// Mitsubishi GX Works2 project: PLC_Group10   PLC: FX3G

// global labels: Global1
VAR_GLOBAL
  ST_DAY10 AT X010 : BOOL;  (* מתג פולס בעליה שמטרתו להתחיל את היום *)
  O_Stock AT D1108 : REAL;  (* תפוזים במלאי *)
  P_Stock AT D1112 : REAL;  (* פומלות במלאי *)
  WashFruit AT X002 : BOOL;  (* מתג תחילת שטיפת הפירות *)
END_VAR
VAR_GLOBAL CONSTANT
  TVal : INT := 30;  (* ערך 3 שניות *)
END_VAR
VAR_GLOBAL
  Coil_Timer1 AT TC3 : BOOL;  (* טיימר 3 שניות להדלקת נורה Y5 *)
  End_CoilT1 AT TS3 : BOOL;  (* מתג שנפתח לאחר 3 שניות *)
  Start_Wash AT Y005 : BOOL;  (* נורה עבור תחילת שלב השטיפה *)
  C_WashM AT D1116 : REAL;  (* קלמנטינות בכלי שטיפה *)
END_VAR
VAR_GLOBAL CONSTANT
  Const05 : REAL := 0.5;  (* קבוע 0.5 להכפלת כמות התפוזים על פי תנאי לתחילת עבודה *)
END_VAR
VAR_GLOBAL
  End_Day AT M7 : BOOL;  (* משתנה נורת עזר 7-סיום עבודה *)
  All_Day_On AT Y010 : BOOL;  (* נורה שדולקת לאורך כל היום *)
END_VAR
VAR_GLOBAL CONSTANT
  Zero : REAL;  (* קבוע אפס *)
END_VAR
VAR_GLOBAL
  Val_Bool AT M1 : BOOL;  (* נורת חיווי שבודקת אם הקלט הוא אפס *)
  Validation_Check AT M0 : BOOL;  (* נורת חיווי תחילת הרצה *)
  O_WashM AT D1118 : REAL;  (* תפוזים בכלי שטיפה *)
  P_WashM AT D1120 : REAL;  (* פומלות בכלי שטיפה *)
END_VAR
VAR_GLOBAL CONSTANT
  Const2 : INT := 2;  (* בדיקת כמות תפוזים *)
END_VAR
VAR_GLOBAL
  Can_Start_Valid AT M8 : BOOL;  (* בדיקת כמות תפוזים במלאי *)
  Start_3sec AT M9 : BOOL;  (* נורת חיווי תחילת טיימר 3 שניות *)
  Half_Oranges AT D1126 : REAL;  (* חצי מכמות התפוזים במלאי *)
END_VAR
VAR_GLOBAL CONSTANT
  Max_Orange100 : INT := 100;  (* כמות מקסימלית של תפוזים בשטיפה *)
END_VAR
VAR_GLOBAL
  Orange_AmountInWash AT D1128 : REAL;  (* כמות התפוזים לשטיפה *)
  Start_Check AT X003 : BOOL;  (* מתג תחילת בדיקת איכות מיץ *)
  Start_Sq AT X001 : BOOL;  (* תחילת סחיטת הפירות *)
  Sq_Light AT Y001 : BOOL;  (* נורת סחיטת הפירות *)
  allToSq AT D1130 : REAL;  (* העברת פירות למיכל סחיטה *)
  Sq_Tank AT D1132 : REAL;  (* מיכל סחיטת הפירות *)
  Moved_To_Sq AT M12 : BOOL;  (* הפירות הועברו למיכל הסחיטה *)
END_VAR
VAR_GLOBAL CONSTANT
  C_Wash_Reset : REAL;  (* איפוס מיכל השטיפה של הקלמנטינות *)
  O_Wash_Reset : REAL;  (* איפוס מיכל השטיפה של התפוזים *)
  P_Wash_Reset : REAL;  (* איפוס מיכל השטיפה של הפומלות *)
END_VAR
VAR_GLOBAL
  Moved_To_Wash AT M13 : BOOL;  (* סיום העברת הפירות למיכלי השטיפה *)
  Sq_LightM AT M14 : BOOL;  (* חיווי נורת סחיטת הפירות *)
  P_C_Wash_Amount AT D1110 : REAL;  (* מספר קלמנטינות ופומלות שיעבור למיכל השטיפה *)
  O_InWash AT M17 : BOOL;  (* חיווי של מספר התפוזים לשטיפה *)
  Min_P_C AT M16 : BOOL;  (* כמות הקלנטינות והפומלות שיכנסו למיכל השטיפה *)
  Min_O AT M15 : BOOL;  (* כמות התפוזים שיכנסו למיכל השטיפה *)
  Stop_SqLight AT M11 : BOOL;  (* כיבוי נורת סחיטת הפירות *)
  Start_3sec_Sq AT X011 : BOOL;  (* מתג הדלקת הבהוב 3 שניות *)
  Click_Twice AT CC1 : BOOL;  (* מונה אירועים שמחכה לשתי לחיצות על מתג איקס 11 *)
END_VAR
VAR_GLOBAL CONSTANT
  Counter_2Clicks : INT := 2;  (* 2לחיצות על איקס 11 *)
END_VAR
VAR_GLOBAL
  Timer_All_Sq AT TC36 : BOOL;  (* טיימר סחיטת פירות למשך 3שניות *)
END_VAR
VAR_GLOBAL CONSTANT
  Val_3Sec : INT := 30;  (* טיימר עובד למשך 3 שניות *)
END_VAR
VAR_GLOBAL
  End_Counting AT CS1 : BOOL;  (* לאחר 2 לחיצות מתחילה הסחיטה *)
  Reset_Flickering AT M31 : BOOL;  (* משתנה שמאתחל את פונקציית ההבהוב *)
  Timer_Sq_Y2 AT TC30 : BOOL;  (* טיימר סחיטת פירות למשך 3שניות *)
END_VAR
VAR_GLOBAL CONSTANT
  Half_sec : INT := 5;  (* נורה וואי 2 דולקת למשך חצי דקה *)
END_VAR
VAR_GLOBAL
  Start_Y2 AT TS30 : BOOL;  (* הדלקת נורה Y2 *)
  Light_Y2 AT Y002 : BOOL;  (* נורת הבהוב Y2 *)
  Timer_Sq_Y3 AT TC32 : BOOL;  (* טיימר שמפעיל את וואי3 שתהבהב *)
  Start_Y3 AT TS32 : BOOL;  (* הדלקת נורה Y3 *)
  Light_Y3 AT Y003 : BOOL;  (* נורת הבהוב Y3 *)
  Stop_Timer_3Sec AT TS36 : BOOL;  (* מפסיק הבהוב לאחר 3 שניות *)
  Juice_Cont AT D4000 : REAL;  (* מיכל מיץ *)
  Moved_To_Juice AT M37 : BOOL;  (* הועברו הפירות הסחוטים למיכל המיץ *)
  Start_Read_Analog AT M40 : BOOL;  (* נורת עזר- יכול לבדוק את הקלט האנלוגי *)
  Analog_Input2 AT D8281 : INT;  (* האינפוט האנלוגי *)
  Analog_Value AT D8291 : REAL;  (* הערך האנאלוגי *)
END_VAR
VAR_GLOBAL CONSTANT
  Const01 : REAL := 1.0;  (* קבוע 1- חסם תחתון לבדיקת איכות תקינה *)
END_VAR
VAR_GLOBAL
  Counting_Input AT CC2 : BOOL;  (* סופר מספר ניסיונות לקלט *)
END_VAR
VAR_GLOBAL CONSTANT
  Two_Inputs : INT := 2;  (* 2 אופצית להכנסת קלט *)
END_VAR
VAR_GLOBAL
  Two_Invalid_Counted AT CS2 : BOOL;  (* נספרו 2 קלטים מחוץ לטווח *)
  Start_5sec AT M42 : BOOL;  (* נורת חיווי תחילת טיימר 5 שניות *)
  Coil_Timer_5sec AT TC34 : BOOL;  (* Y4 תדלוק למשך 5 שניות *)
END_VAR
VAR_GLOBAL CONSTANT
  T_Value_5sec : INT := 50;  (* ערך 5 שניות *)
END_VAR
VAR_GLOBAL
  Finished_5sec AT M43 : BOOL;  (* נורת עזר- סיום 5 שניות *)
  End_CoilT2 AT TS34 : BOOL;  (* מתג שנפתח לאחר 5 שניות *)
  Finish_Qcheck AT Y004 : BOOL;  (* נורה שבדיקת האיכות בוצעה בהצלחה *)
  Storage_Cont AT D4002 : REAL;  (* מיכל אחסון *)
  Moved_To_Storage AT M44 : BOOL;  (* הועבר המיץ למיכל האחסון *)
  Empty_Sq_Tank AT M45 : BOOL;  (* המיץ הועבר ממיכל הסחיטה למיכל המיץ *)
END_VAR
VAR_GLOBAL CONSTANT
  Convert_Analog : REAL := 404.5;  (* המרת ערך אנאלוגי מהבקר למחשב *)
  Const5 : REAL := 5.0;  (* קבוע 5 *)
END_VAR
VAR_GLOBAL
  Input_Not_In_Range_1 AT M5 : BOOL;  (* נורת עזר- הקלט האנלוגי לא בטווח- קטן מ1 *)
  Input_Not_In_Range_5 AT M6 : BOOL;  (* נורת עזר- הקלט האנלוגי לא בטווח- גדול מ5 *)
  M_Start_Check AT M3 : BOOL;  (* נורת חיווי שמתג X3 הופעל *)
  Input_In_Range AT M4 : BOOL;  (* נורת עזר- הקלט האנלוגי בטווח *)
  End_Day_007 AT X007 : BOOL;  (* מתג סיום יום העבודה *)
  Not_In_Range_5 AT M49 : BOOL;  (* הערך גדול מ5 *)
  Not_In_Range_1 AT M47 : BOOL;  (* הערך קטן מ1 *)
  End_Day_Flickering AT TC38 : BOOL;  (* תחילת הבהוב סיום יום העבודה *)
  Flickering_End_Day AT TC40 : BOOL;  (* הבהוב סוף יום *)
  End_3Sec_End_Day AT TS38 : BOOL;  (* סיום הבהוב 3 שניות סוף יום *)
  End_Half_Sec AT TS40 : BOOL;  (* סיום חצי שניה של הבהוב *)
  Start_Half_Sec AT M50 : BOOL;  (* תחילת חצי שניה *)
  Continue_To_Blink AT M51 : BOOL;  (* המשך הבהוב *)
  Help_Timer_Half_Sec AT TC41 : BOOL;  (* טיימר חצי שניה *)
  Help_End_Half_Sec AT TS41 : BOOL;  (* סיום חצי שניה של הבהוב עזרה *)
  Help_Me AT M52 : BOOL;  (* הצילינינא *)
  Help_Me_2 AT M53 : BOOL;  (* הצילינינא2 *)
  No_More AT M55 : BOOL;  (* סיום עבודה *)
END_VAR
VAR_GLOBAL CONSTANT
  Const_4 : REAL := 4.0;  (* קבוע 4- כמות מיץ מינימלית להמשך תהליך *)
END_VAR
VAR_GLOBAL
  Move_To_Filter AT M56 : BOOL;  (* נורת עזר- 4 ליטר מיץ הועבר למיכל הסינון *)
  Juice_To_Filter AT D1102 : REAL;  (* העברת 4 ליטר מיץ למיכל סינון *)
  Start_Filtering AT X000 : BOOL;  (* מתג שמתחיל את שלב הסינון *)
  Juice_Filtered AT D1124 : REAL;  (* מיכל מיץ מסונן *)
  Storage_Filtered AT M57 : BOOL;  (* נורת עזר- הורדת המיץ המסונן מהאחסון *)
  Aperol_Spritz AT D4004 : REAL;  (* אפרול שפריץ- המיץ המסונן האלכוהולי שלנו *)
  Analog_Output AT D8282 : INT;  (* האאוטפוט האנלוגי *)
  Filtering_Time AT Y000 : BOOL;  (* נורה שדולקת בכל תהליך הסינון *)
END_VAR
VAR_GLOBAL CONSTANT
  Two_Liter_Alcohol : REAL := 2.0;  (* הוספת 2 ליטר אלכוהול למיץ המסונן *)
END_VAR
VAR_GLOBAL
  Aperol_To_Taste AT Y006 : BOOL;  (* נורה שנדלקת כשהאפרול מוכן *)
  Counting_Rates AT CC3 : BOOL;  (* סופר 4 ציונים *)
END_VAR
VAR_GLOBAL CONSTANT
  Four_Rates : INT := 4;  (* 4 ציונים *)
END_VAR
VAR_GLOBAL
  Four_Rates_Given AT CS3 : BOOL;  (* ניתנו 4 ציונים *)
  Start_Rating AT X005 : BOOL;  (* מתג שמתחיל קליטת ציון *)
  M_Start_Check_Rate AT M10 : BOOL;  (* נורת חיווי ניתן ציון *)
  Read_Analog_Rate AT M18 : BOOL;  (* נורת עזר- יכול לבדוק את הקלט האנלוגי *)
  Analog_Value_Rate AT D8293 : REAL;  (* הערך האנאלוגי *)
  Total_Rates AT D1114 : REAL;  (* סך הציונים *)
  Average_Grade AT D1106 : INT;  (* הציון הממוצע של המשקה *)
  Final_Grade AT M59 : BOOL;  (* חושב ציון סופי למשקה *)
  Analog_Input1 AT D8280 : INT;  (* האינפוט האנלוגי *)
  Analog_Showed AT M30 : BOOL;  (* הציון נמצאבOUTPUT *)
  Total_Rates_W AT D1122 : INT;  (* סך הציונים בWORLD *)
  End_Filtering_Light AT TS50 : BOOL;  (* סיום נורת הסינון *)
  Start_Filtering_Light AT TC50 : BOOL;  (* מתג שמתחיל את שלב הסינון *)
  Drink_Is_Ready AT M28 : BOOL;  (* המשקה האלכוהולי מוכן! *)
  Drink_Timer AT TC60 : BOOL;  (* טיימר משקה הוכן *)
END_VAR
VAR_GLOBAL CONSTANT
  Four_Sec : INT := 40;  (* 4 שניות *)
END_VAR
VAR_GLOBAL
  Moved_From_Storage AT M26 : BOOL;  (* העברה 4 מהאחסון לסינון *)
  Average_Output AT D1134 : INT;  (* ממוצע להצגה לאאוטפוט *)
  Output_Convert AT M32 : BOOL;  (* המרה לאאוטפוט *)
  Grade_Added AT M39 : BOOL;  (* נוסף ציון *)
  Lets_Get_Wasted AT M46 : BOOL;  (* יאללה פארטי *)
END_VAR
VAR_GLOBAL CONSTANT
  Const400 : INT := 400;  (* הכפלת אפרול שפריץ בקבוע בשביל שיוציא באנלוג אאוטפוט *)
END_VAR
VAR_GLOBAL
  If_Fruits_Ended AT M24 : BOOL;  (* נגמר סוג אחד או יותר של פרי *)
  Drink_Timer_Ended AT TS60 : BOOL;  (* סיום טיימר נורת ערבוב *)
  Start_Again AT M60 : BOOL;  (* סיום יום והתחלת יום חדש *)
  Did_You_Get_True AT M88 : BOOL;  (* נורה שבודקת שעבר זרם דרך בדיקת שני תפוזים *)
  End_Day_Bulb AT M70 : BOOL;  (* מתג סיום יום העבודה *)
  C_Stock AT D4006 : REAL;  (* קלמנטינות במלאי *)
  Damaged_Juice AT M73 : BOOL;  (* מיץ לא תקין *)
END_VAR

// task Task_01 (event TRUE, interval 0, priority 31): POU_01

PROGRAM POU_01
VAR
  O_output : REAL;
  C_output : REAL;
  P_output : REAL;
  Start_Flickering : BOOL;  (* תחילת שלב הסחיטה- ההבהוב *)
  Move_To : BOOL;
END_VAR
(* structured ladder/FBD written out as ST: instructions are called as NAME(EN, inputs, outputs); _pN, _eN, _tN stand for wires *)
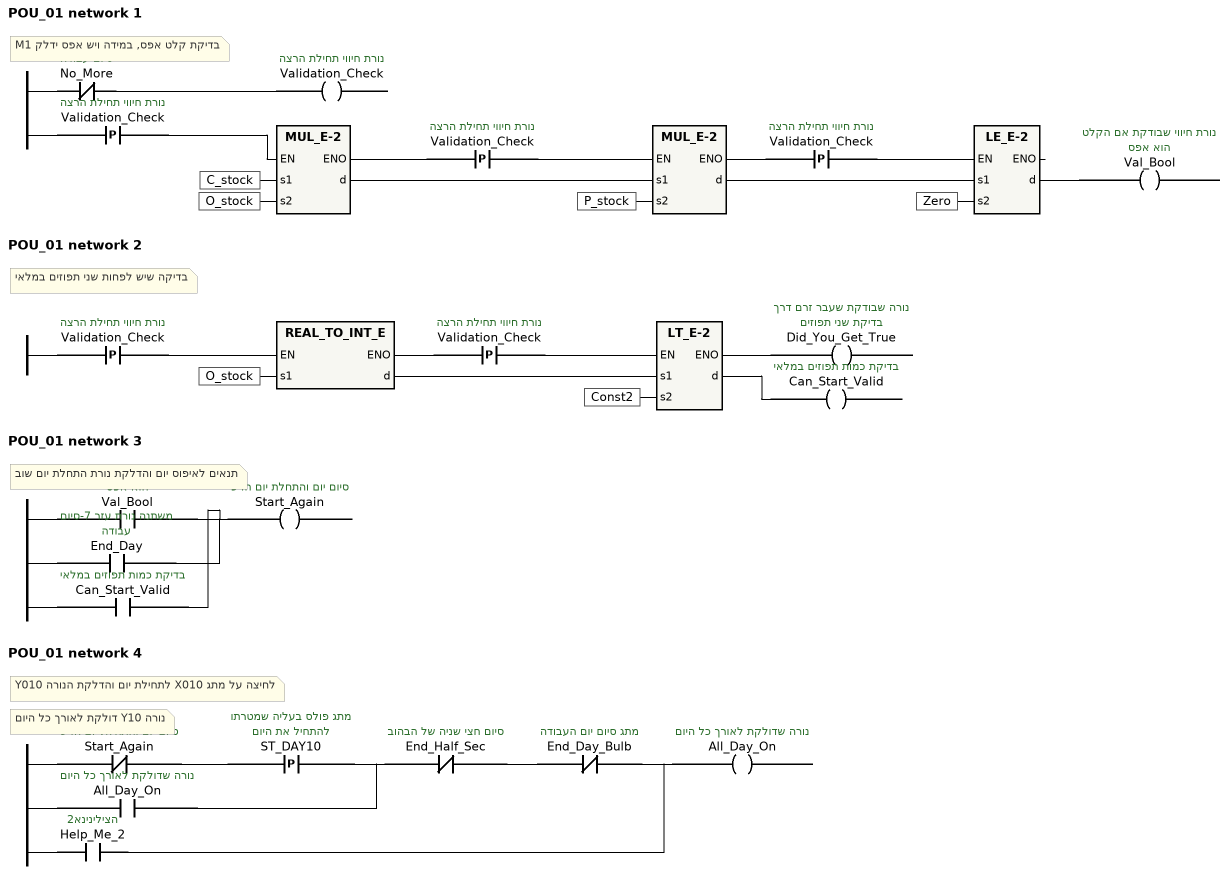
(* network 1 *)
(* בדיקת קלט אפס, במידה ויש אפס ידלק M1 *)
Validation_Check := NOT No_More;
_e2 := MUL_E(LDP(TRUE, Validation_Check), C_stock, O_stock, _t1);
_e4 := MUL_E(_e2 AND LDP(TRUE, Validation_Check), _t1, P_stock, _t3);
LE_E(_e4 AND LDP(TRUE, Validation_Check), _t3, Zero, _t5);
Val_Bool := _t5;
(* network 2 *)
(* בדיקה שיש לפחות שני תפוזים במלאי *)
_e2 := REAL_TO_INT_E(LDP(TRUE, Validation_Check), O_stock, _t1);
_e4 := LT_E(_e2 AND LDP(TRUE, Validation_Check), _t1, Const2, _t3);
Did_You_Get_True := _e4;
Can_Start_Valid := _t3;
(* network 3 *)
(* תנאים לאיפוס יום והדלקת נורת התחלת יום שוב *)
Start_Again := Val_Bool OR End_Day OR Can_Start_Valid;
(* network 4 *)
(* לחיצה על מתג X010 לתחילת יום והדלקת הנורה Y010 *)
(* נורה Y10 דולקת לאורך כל היום *)
All_Day_On := ((((NOT Start_Again AND LDP(TRUE, ST_DAY10)) OR All_Day_On) AND NOT End_Half_Sec) AND NOT End_Day_Bulb) OR Help_Me_2;
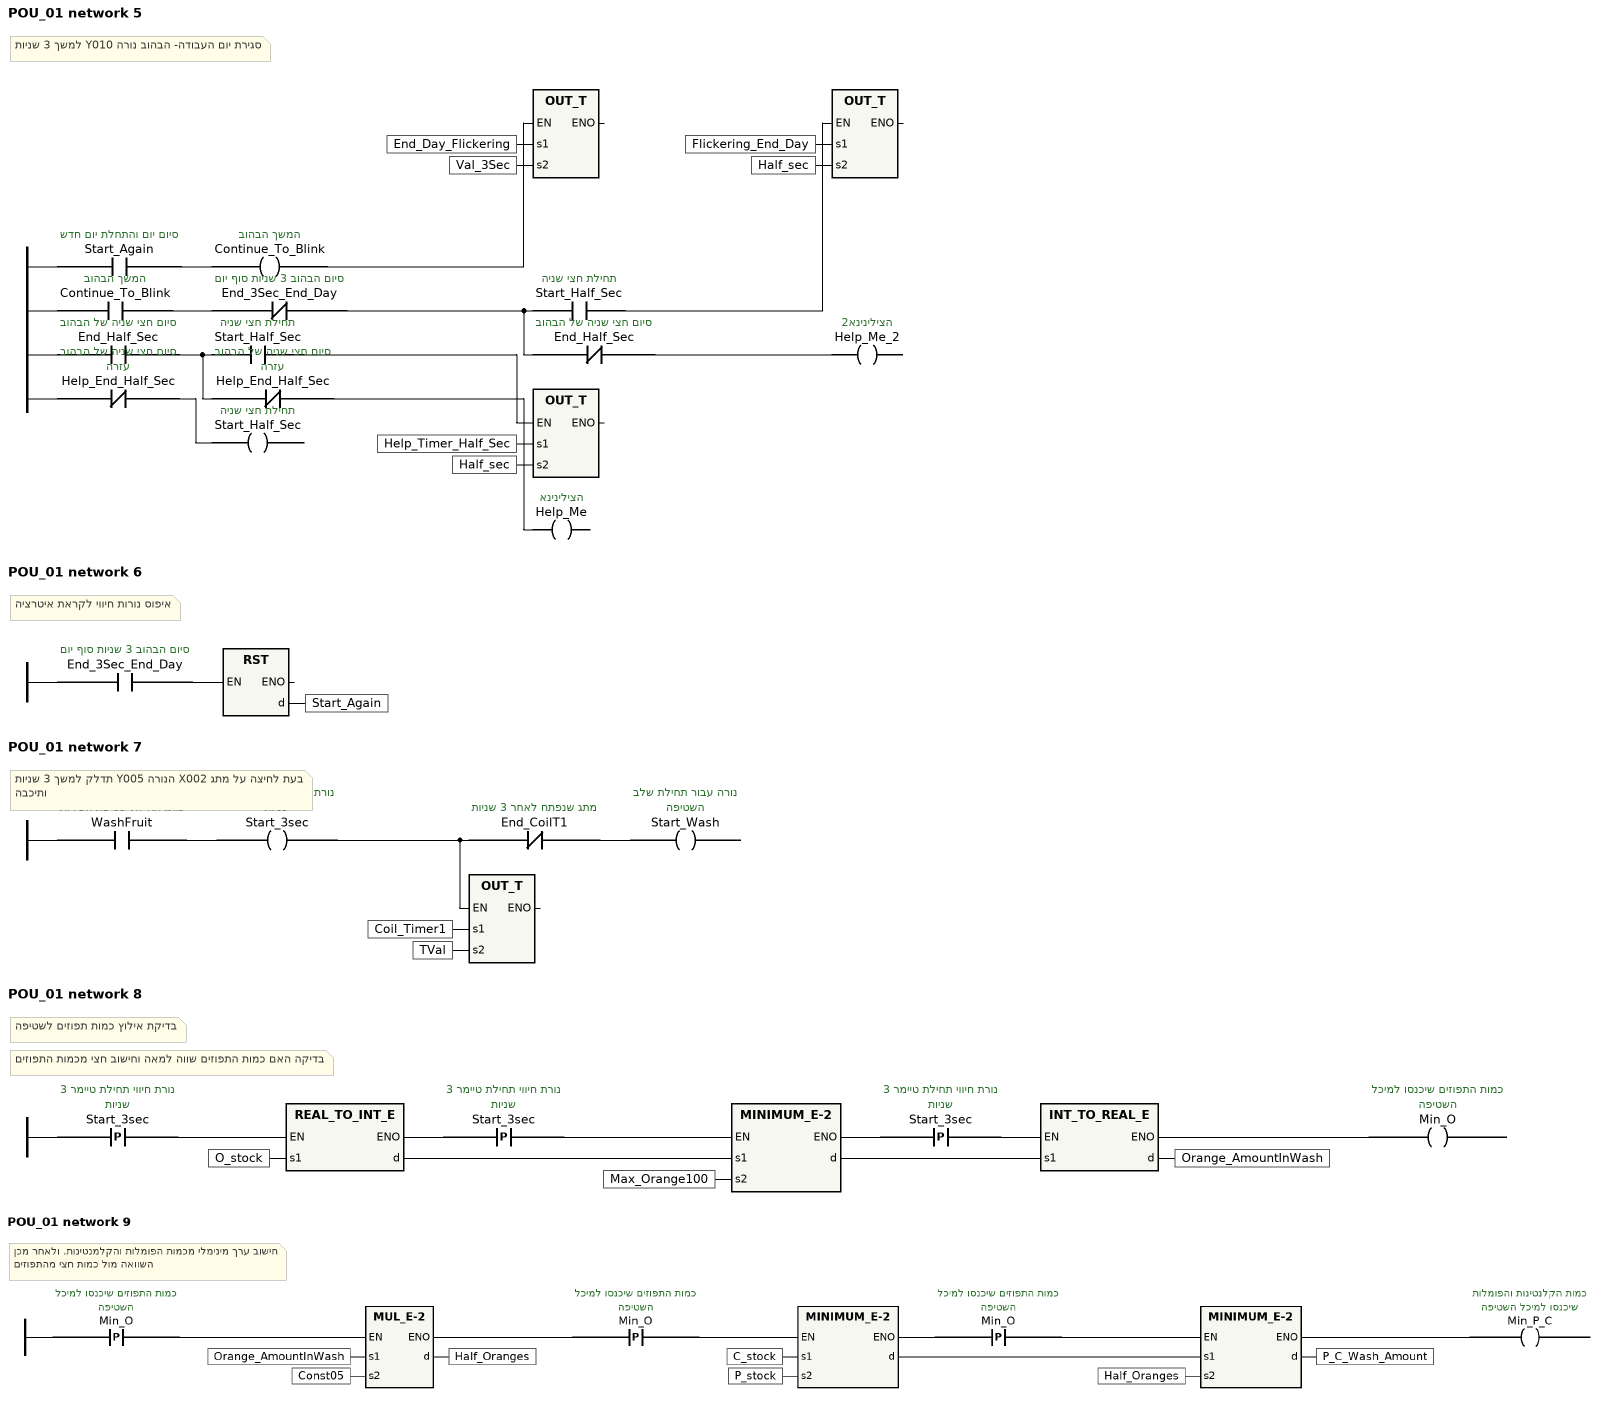
(* network 5 *)
(* סגירת יום העבודה- הבהוב נורה Y010 למשך 3 שניות *)
Continue_To_Blink := Start_Again;
OUT_T(Start_Again, End_Day_Flickering, Val_3Sec);
_p1 := Continue_To_Blink AND NOT End_3Sec_End_Day;
OUT_T(_p1 AND Start_Half_Sec, Flickering_End_Day, Half_sec);
Help_Me_2 := _p1 AND NOT End_Half_Sec;
OUT_T(End_Half_Sec AND Start_Half_Sec, Help_Timer_Half_Sec, Half_sec);
Help_Me := End_Half_Sec AND NOT Help_End_Half_Sec;
Start_Half_Sec := NOT Help_End_Half_Sec;
(* network 6 *)
(* איפוס נורות חיווי לקראת איטרציה *)
RST(End_3Sec_End_Day, Start_Again);
(* network 7 *)
(* בעת לחיצה על מתג X002 הנורה Y005 תדלק למשך 3 שניות ותיכבה *)
Start_3sec := WashFruit;
Start_Wash := WashFruit AND NOT End_CoilT1;
OUT_T(WashFruit, Coil_Timer1, TVal);
(* network 8 *)
(* בדיקת אילוץ כמות תפוזים לשטיפה *)
(* בדיקה האם כמות התפוזים שווה למאה וחישוב חצי מכמות התפוזים *)
_e2 := REAL_TO_INT_E(LDP(TRUE, Start_3sec), O_stock, _t1);
_e4 := MINIMUM_E(_e2 AND LDP(TRUE, Start_3sec), _t1, Max_Orange100, _t3);
_e5 := INT_TO_REAL_E(_e4 AND LDP(TRUE, Start_3sec), _t3, Orange_AmountInWash);
Min_O := _e5;
(* network 9 *)
(* חישוב ערך מינימלי מכמות הפומלות והקלמנטינות. ולאחר מכן השוואה מול כמות חצי מהתפוזים *)
_e1 := MUL_E(LDP(TRUE, Min_O), Orange_AmountInWash, Const05, Half_Oranges);
_e3 := MINIMUM_E(_e1 AND LDP(TRUE, Min_O), C_stock, P_stock, _t2);
_e4 := MINIMUM_E(_e3 AND LDP(TRUE, Min_O), _t2, Half_Oranges, P_C_Wash_Amount);
Min_P_C := _e4;
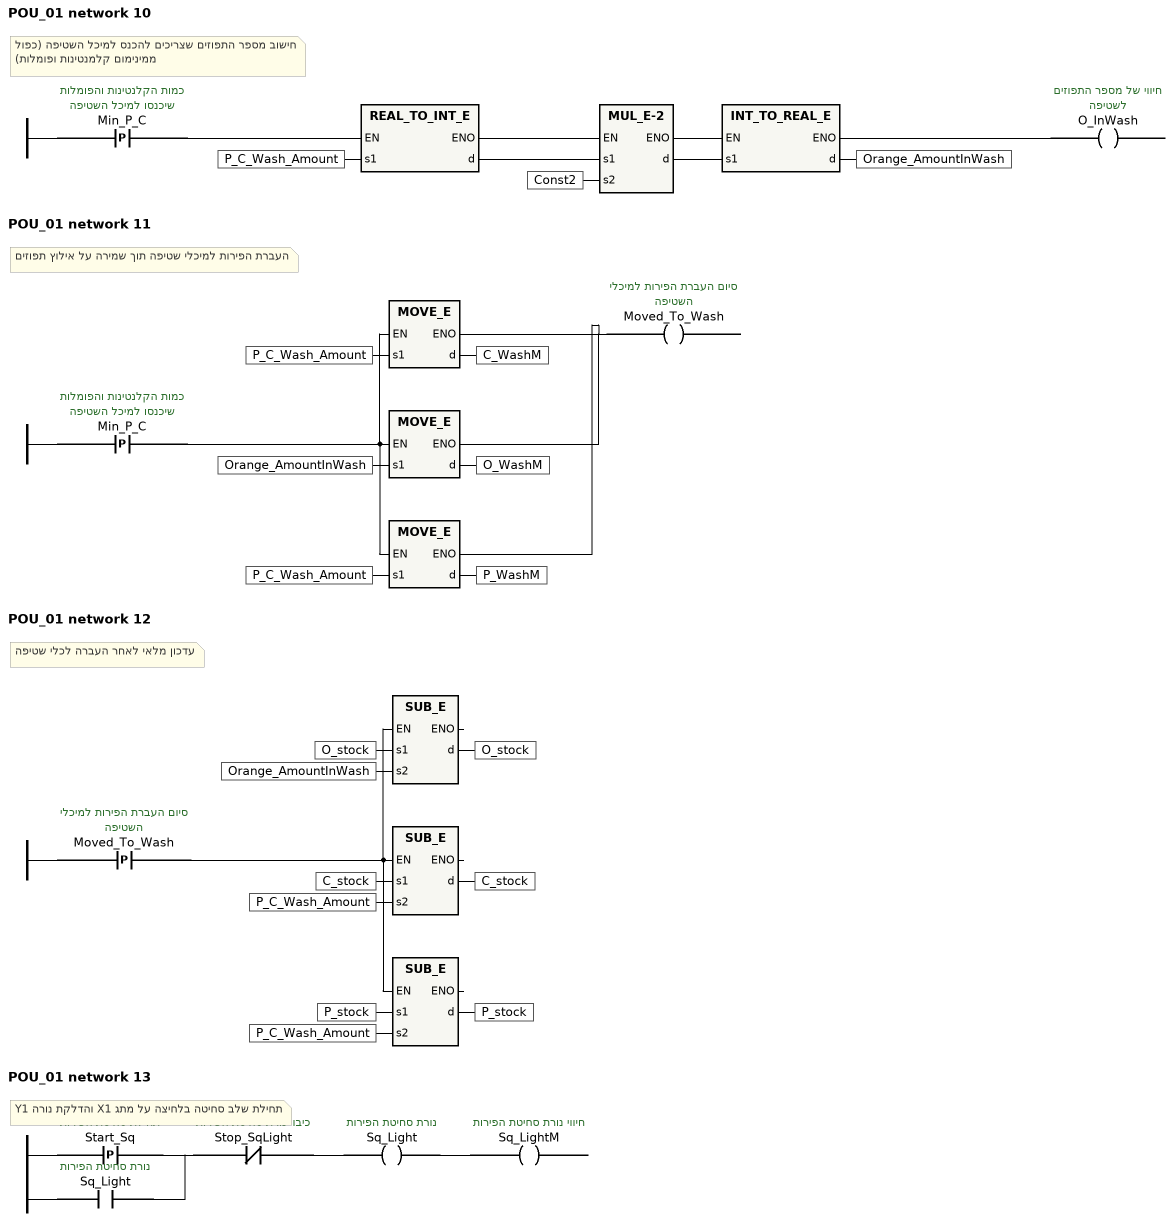
(* network 10 *)
(* חישוב מספר התפוזים שצריכים להכנס למיכל השטיפה (כפול ממינימום קלמנטינות ופומלות) *)
_e2 := REAL_TO_INT_E(LDP(TRUE, Min_P_C), P_C_Wash_Amount, _t1);
_e4 := MUL_E(_e2, _t1, Const2, _t3);
_e5 := INT_TO_REAL_E(_e4, _t3, Orange_AmountInWash);
O_InWash := _e5;
(* network 11 *)
(* העברת הפירות למיכלי שטיפה תוך שמירה על אילוץ תפוזים *)
_p1 := LDP(TRUE, Min_P_C);
_e2 := MOVE_E(_p1, P_C_Wash_Amount, C_WashM);
_e3 := MOVE_E(_p1, Orange_AmountInWash, O_WashM);
_e4 := MOVE_E(_p1, P_C_Wash_Amount, P_WashM);
Moved_To_Wash := _e2 OR _e3 OR _e4;
(* network 12 *)
(* עדכון מלאי לאחר העברה לכלי שטיפה *)
_p1 := LDP(TRUE, Moved_To_Wash);
SUB_E(_p1, O_stock, Orange_AmountInWash, O_stock);
SUB_E(_p1, C_stock, P_C_Wash_Amount, C_stock);
SUB_E(_p1, P_stock, P_C_Wash_Amount, P_stock);
(* network 13 *)
(* תחילת שלב סחיטה בלחיצה על מתג X1 והדלקת נורה Y1 *)
_p1 := (LDP(TRUE, Start_Sq) OR Sq_Light) AND NOT Stop_SqLight;
Sq_Light := _p1;
Sq_LightM := _p1;
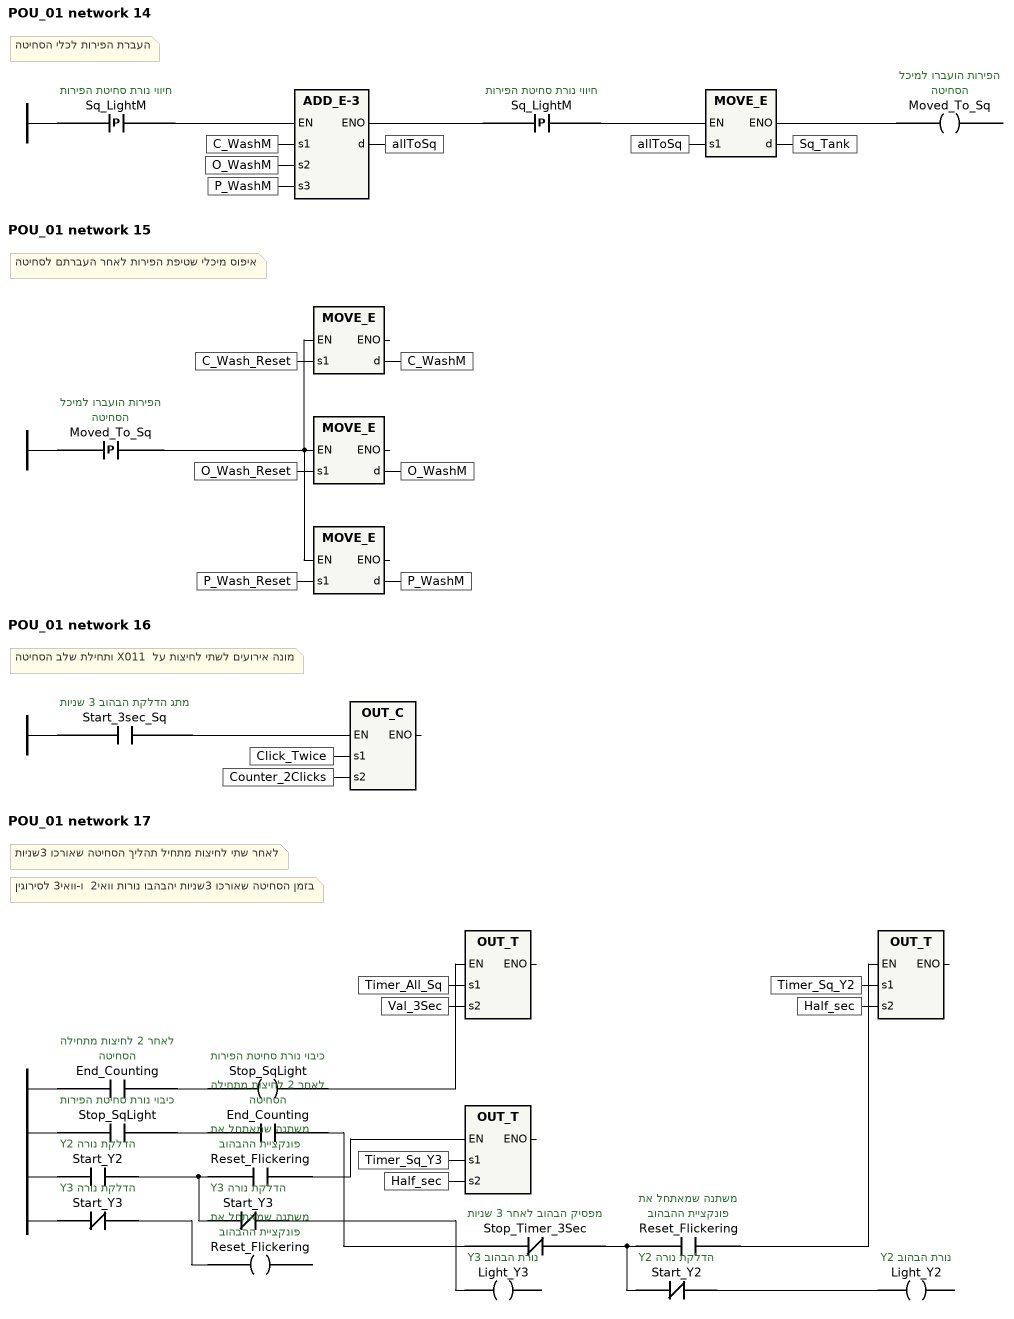
(* network 14 *)
(* העברת הפירות לכלי הסחיטה *)
_e1 := ADD_E(LDP(TRUE, Sq_LightM), C_WashM, O_WashM, P_WashM, allToSq);
_e2 := MOVE_E(_e1 AND LDP(TRUE, Sq_LightM), allToSq, Sq_Tank);
Moved_To_Sq := _e2;
(* network 15 *)
(* איפוס מיכלי שטיפת הפירות לאחר העברתם לסחיטה *)
_p1 := LDP(TRUE, Moved_To_Sq);
MOVE_E(_p1, C_Wash_Reset, C_WashM);
MOVE_E(_p1, O_Wash_Reset, O_WashM);
MOVE_E(_p1, P_Wash_Reset, P_WashM);
(* network 16 *)
(* מונה אירועים לשתי לחיצות על  X011 ותחילת שלב הסחיטה *)
OUT_C(Start_3sec_Sq, Click_Twice, Counter_2Clicks);
(* network 17 *)
(* לאחר שתי לחיצות מתחיל תהליך הסחיטה שאורכו 3שניות *)
(* בזמן הסחיטה שאורכו 3שניות יהבהבו נורות וואי2  ו-וואי3 לסירוגין *)
Stop_SqLight := End_Counting;
OUT_T(End_Counting, Timer_All_Sq, Val_3Sec);
_p1 := Stop_SqLight AND End_Counting AND NOT Stop_Timer_3Sec;
OUT_T(_p1 AND Reset_Flickering, Timer_Sq_Y2, Half_sec);
Light_Y2 := _p1 AND NOT Start_Y2;
OUT_T(Start_Y2 AND Reset_Flickering, Timer_Sq_Y3, Half_sec);
Light_Y3 := Start_Y2 AND NOT Start_Y3;
Reset_Flickering := NOT Start_Y3;
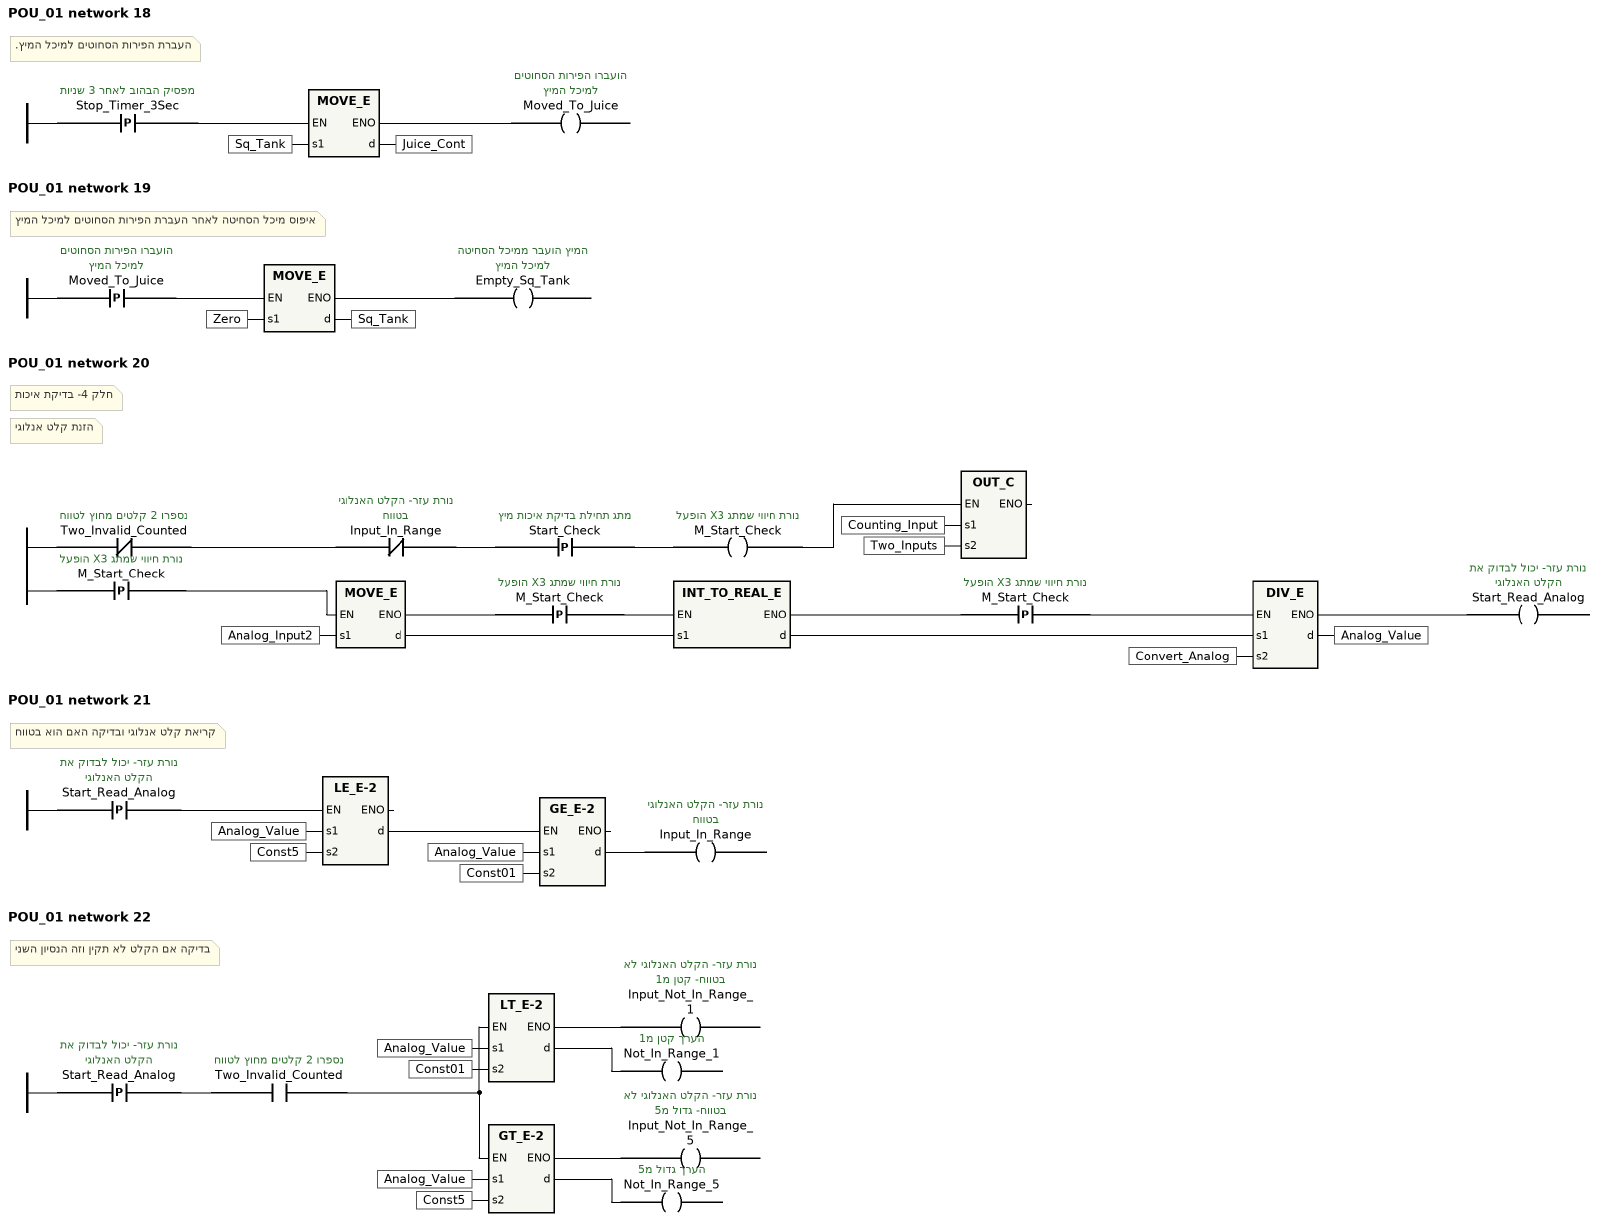
(* network 18 *)
(* העברת הפירות הסחוטים למיכל המיץ. *)
_e1 := MOVE_E(LDP(TRUE, Stop_Timer_3Sec), Sq_Tank, Juice_Cont);
Moved_To_Juice := _e1;
(* network 19 *)
(* איפוס מיכל הסחיטה לאחר העברת הפירות הסחוטים למיכל המיץ *)
_e1 := MOVE_E(LDP(TRUE, Moved_To_Juice), Zero, Sq_Tank);
Empty_Sq_Tank := _e1;
(* network 20 *)
(* חלק 4- בדיקת איכות *)
(* הזנת קלט אנלוגי *)
_p1 := NOT Two_Invalid_Counted AND NOT Input_In_Range AND LDP(TRUE, Start_Check);
M_Start_Check := _p1;
OUT_C(_p1, Counting_Input, Two_Inputs);
_e3 := MOVE_E(LDP(TRUE, M_Start_Check), Analog_Input2, _t2);
_e5 := INT_TO_REAL_E(_e3 AND LDP(TRUE, M_Start_Check), _t2, _t4);
_e6 := DIV_E(_e5 AND LDP(TRUE, M_Start_Check), _t4, Convert_Analog, Analog_Value);
Start_Read_Analog := _e6;
(* network 21 *)
(* קריאת קלט אנלוגי ובדיקה האם הוא בטווח *)
LE_E(LDP(TRUE, Start_Read_Analog), Analog_Value, Const5, _t1);
GE_E(_t1, Analog_Value, Const01, _t2);
Input_In_Range := _t2;
(* network 22 *)
(* בדיקה אם הקלט לא תקין וזה הנסיון השני *)
_p1 := LDP(TRUE, Start_Read_Analog) AND Two_Invalid_Counted;
_e3 := LT_E(_p1, Analog_Value, Const01, _t2);
Input_Not_In_Range_1 := _e3;
Not_In_Range_1 := _t2;
_e5 := GT_E(_p1, Analog_Value, Const5, _t4);
Input_Not_In_Range_5 := _e5;
Not_In_Range_5 := _t4;
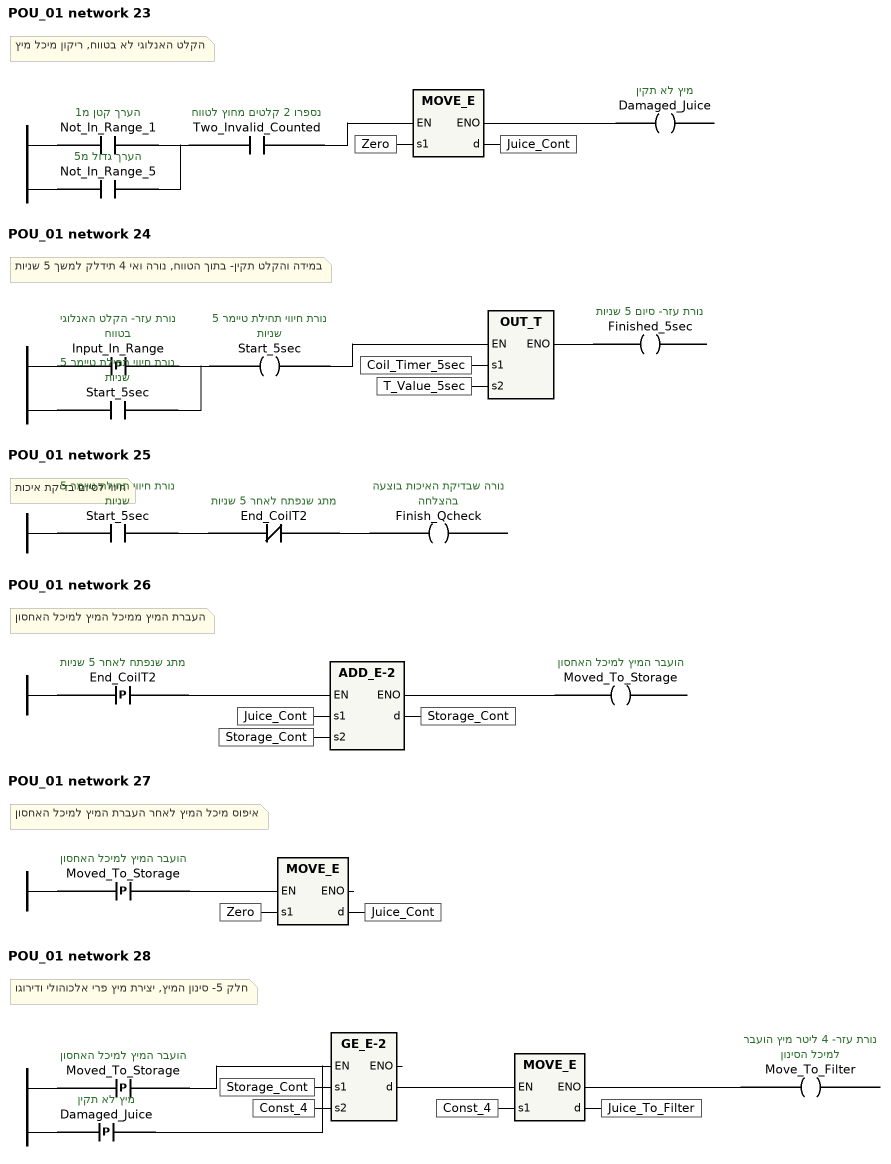
(* network 23 *)
(* הקלט האנלוגי לא בטווח, ריקון מיכל מיץ *)
_e1 := MOVE_E((Not_In_Range_1 OR Not_In_Range_5) AND Two_Invalid_Counted, Zero, Juice_Cont);
Damaged_Juice := _e1;
(* network 24 *)
(* במידה והקלט תקין- בתוך הטווח, נורה ואי 4 תידלק למשך 5 שניות *)
_p1 := LDP(TRUE, Input_In_Range) OR Start_5sec;
Start_5sec := _p1;
_e2 := OUT_T(_p1, Coil_Timer_5sec, T_Value_5sec);
Finished_5sec := _e2;
(* network 25 *)
(* חיווי לסיום בדיקת איכות *)
Finish_Qcheck := Start_5sec AND NOT End_CoilT2;
(* network 26 *)
(* העברת המיץ ממיכל המיץ למיכל האחסון *)
_e1 := ADD_E(LDP(TRUE, End_CoilT2), Juice_Cont, Storage_Cont, Storage_Cont);
Moved_To_Storage := _e1;
(* network 27 *)
(* איפוס מיכל המיץ לאחר העברת המיץ למיכל האחסון *)
MOVE_E(LDP(TRUE, Moved_To_Storage), Zero, Juice_Cont);
(* network 28 *)
(* חלק 5- סינון המיץ, יצירת מיץ פרי אלכוהולי ודירוגו *)
GE_E(LDP(TRUE, Moved_To_Storage) OR LDP(TRUE, Damaged_Juice), Storage_Cont, Const_4, _t1);
_e2 := MOVE_E(_t1, Const_4, Juice_To_Filter);
Move_To_Filter := _e2;
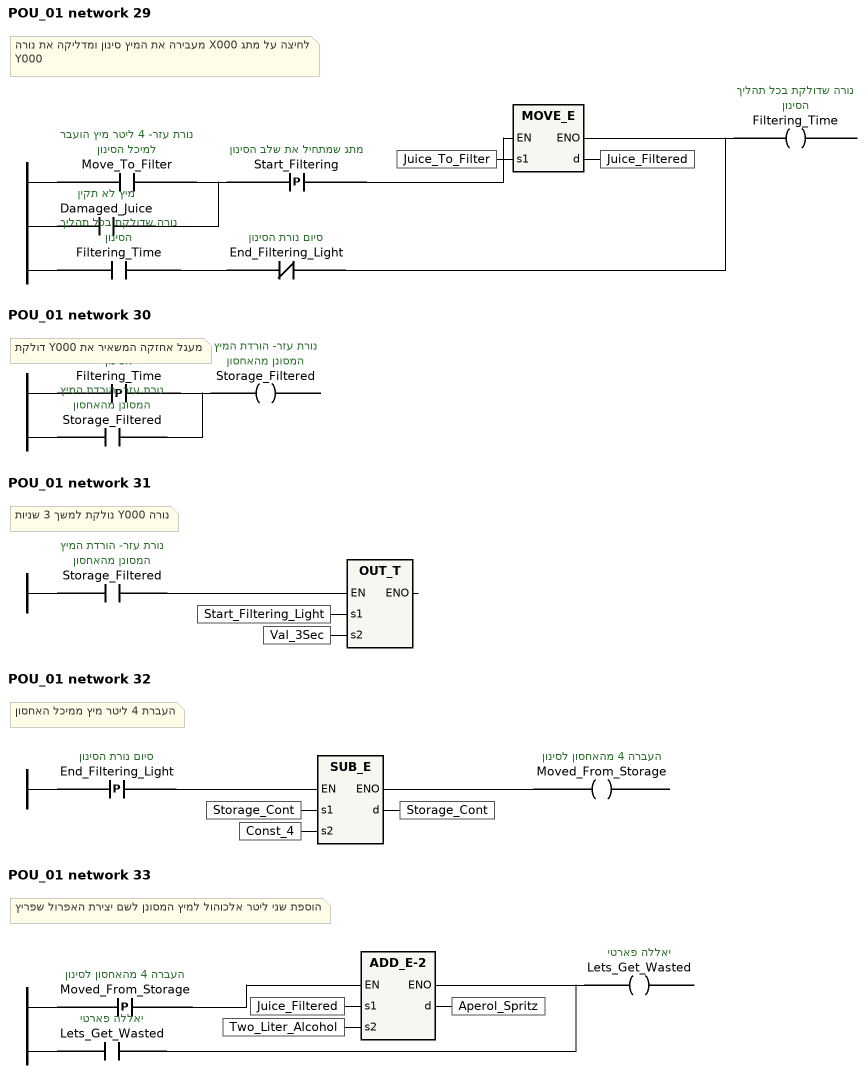
(* network 29 *)
(* לחיצה על מתג X000 מעבירה את המיץ סינון ומדליקה את נורה Y000 *)
_e1 := MOVE_E((Move_To_Filter OR Damaged_Juice) AND LDP(TRUE, Start_Filtering), Juice_To_Filter, Juice_Filtered);
Filtering_Time := _e1 OR (Filtering_Time AND NOT End_Filtering_Light);
(* network 30 *)
(* מעגל אחזקה המשאיר את Y000 דולקת *)
Storage_Filtered := LDP(TRUE, Filtering_Time) OR Storage_Filtered;
(* network 31 *)
(* נורה Y000 נולקת למשך 3 שניות *)
OUT_T(Storage_Filtered, Start_Filtering_Light, Val_3Sec);
(* network 32 *)
(* העברת 4 ליטר מיץ ממיכל האחסון *)
_e1 := SUB_E(LDP(TRUE, End_Filtering_Light), Storage_Cont, Const_4, Storage_Cont);
Moved_From_Storage := _e1;
(* network 33 *)
(* הוספת שני ליטר אלכוהול למיץ המסונן לשם יצירת האפרול שפריץ *)
_e1 := ADD_E(LDP(TRUE, Moved_From_Storage), Juice_Filtered, Two_Liter_Alcohol, Aperol_Spritz);
Lets_Get_Wasted := _e1 OR Lets_Get_Wasted;
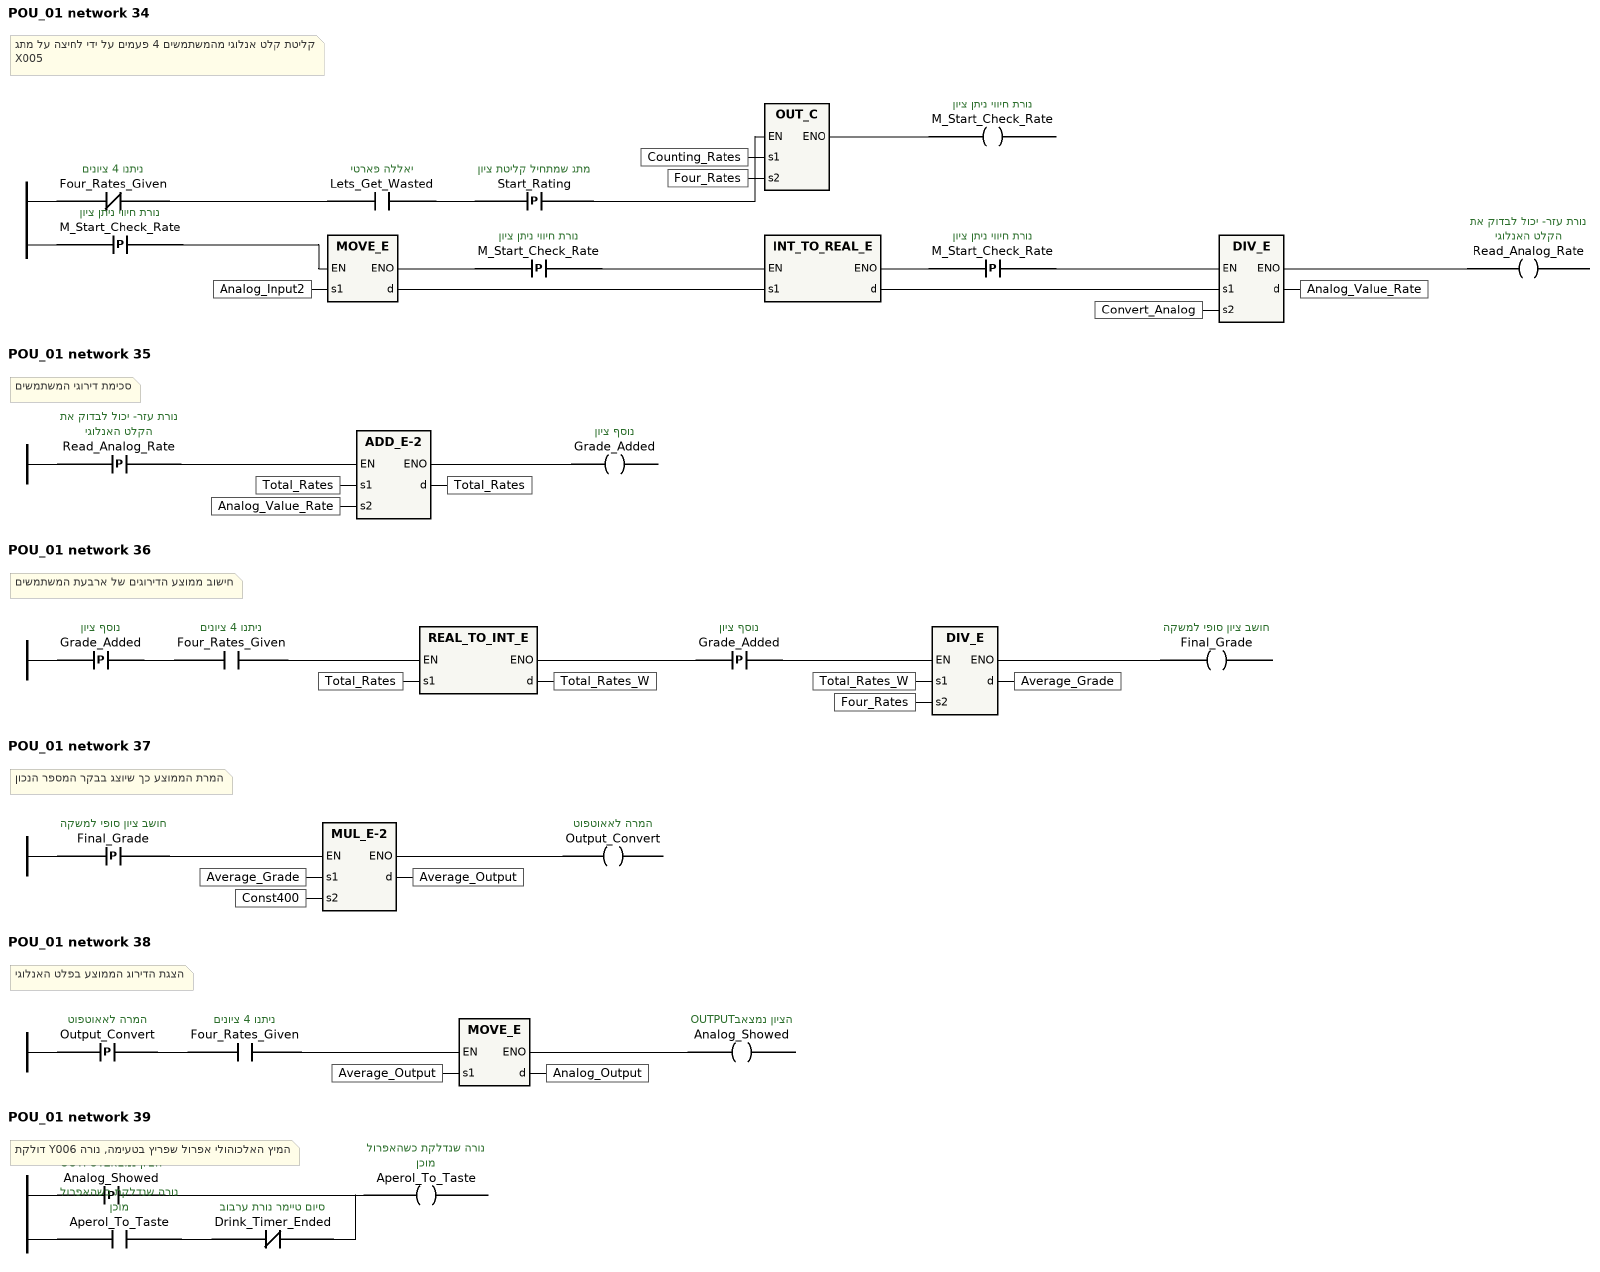
(* network 34 *)
(* קליטת קלט אנלוגי מהמשתמשים 4 פעמים על ידי לחיצה על מתג X005 *)
_e1 := OUT_C(NOT Four_Rates_Given AND Lets_Get_Wasted AND LDP(TRUE, Start_Rating), Counting_Rates, Four_Rates);
M_Start_Check_Rate := _e1;
_e3 := MOVE_E(LDP(TRUE, M_Start_Check_Rate), Analog_Input2, _t2);
_e5 := INT_TO_REAL_E(_e3 AND LDP(TRUE, M_Start_Check_Rate), _t2, _t4);
_e6 := DIV_E(_e5 AND LDP(TRUE, M_Start_Check_Rate), _t4, Convert_Analog, Analog_Value_Rate);
Read_Analog_Rate := _e6;
(* network 35 *)
(* סכימת דירוגי המשתמשים *)
_e1 := ADD_E(LDP(TRUE, Read_Analog_Rate), Total_Rates, Analog_Value_Rate, Total_Rates);
Grade_Added := _e1;
(* network 36 *)
(* חישוב ממוצע הדירוגים של ארבעת המשתמשים *)
_e1 := REAL_TO_INT_E(LDP(TRUE, Grade_Added) AND Four_Rates_Given, Total_Rates, Total_Rates_W);
_e2 := DIV_E(_e1 AND LDP(TRUE, Grade_Added), Total_Rates_W, Four_Rates, Average_Grade);
Final_Grade := _e2;
(* network 37 *)
(* המרת הממוצע כך שיוצג בבקר המספר הנכון *)
_e1 := MUL_E(LDP(TRUE, Final_Grade), Average_Grade, Const400, Average_Output);
Output_Convert := _e1;
(* network 38 *)
(* הצגת הדירוג הממוצע בפלט האנלוגי *)
_e1 := MOVE_E(LDP(TRUE, Output_Convert) AND Four_Rates_Given, Average_Output, Analog_Output);
Analog_Showed := _e1;
(* network 39 *)
(* המיץ האלכוהולי אפרול שפריץ בטעימה, נורה Y006 דולקת *)
Aperol_To_Taste := LDP(TRUE, Analog_Showed) OR (Aperol_To_Taste AND NOT Drink_Timer_Ended);
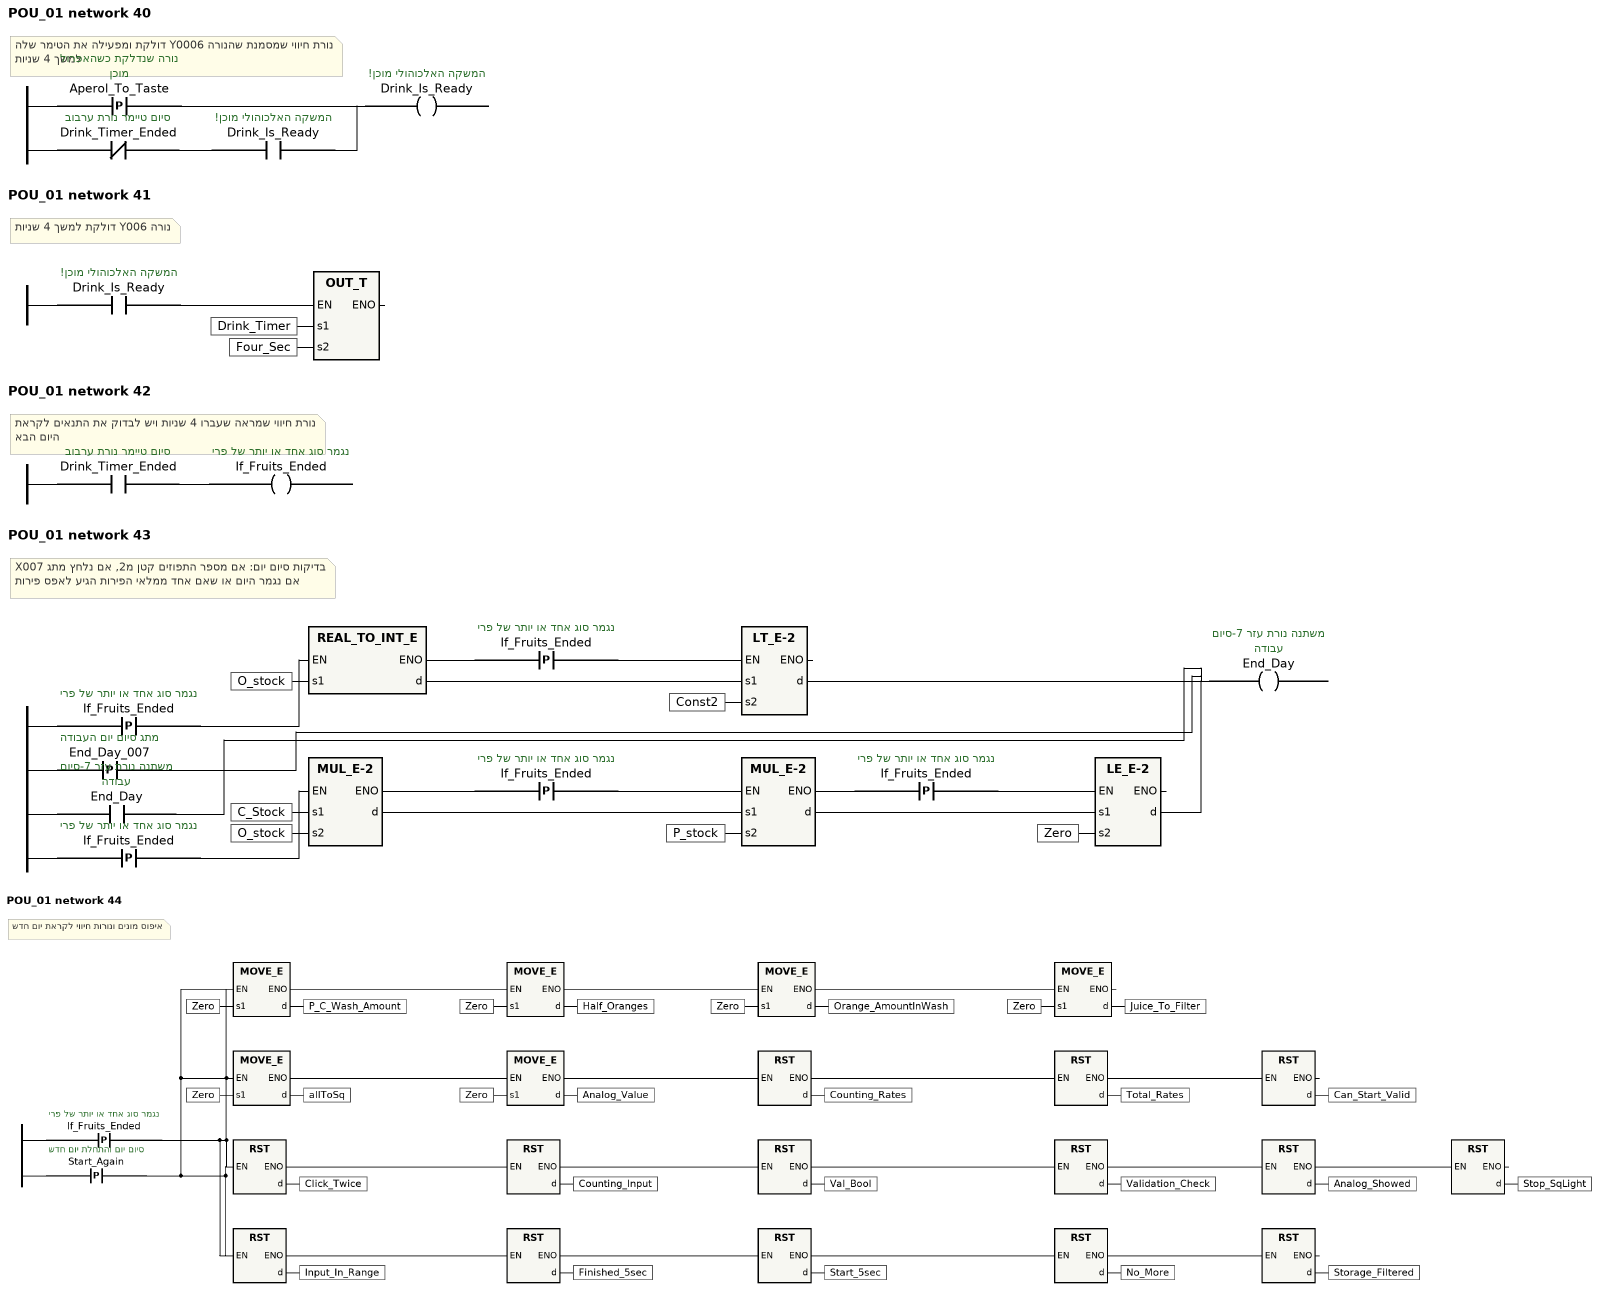
(* network 40 *)
(* נורת חיווי שמסמנת שהנורה Y0006 דולקת ומפעילה את הטימר שלה למשך 4 שניות *)
Drink_Is_Ready := LDP(TRUE, Aperol_To_Taste) OR (NOT Drink_Timer_Ended AND Drink_Is_Ready);
(* network 41 *)
(* נורה Y006 דולקת למשך 4 שניות *)
OUT_T(Drink_Is_Ready, Drink_Timer, Four_Sec);
(* network 42 *)
(* נורת חיווי שמראה שעברו 4 שניות ויש לבדוק את התנאים לקראת היום הבא *)
If_Fruits_Ended := Drink_Timer_Ended;
(* network 43 *)
(* בדיקות סיום יום: אם מספר התפוזים קטן מ2, אם נלחץ מתג X007 אם נגמר היום או שאם אחד ממלאי הפירות הגיע לאפס פירות *)
_e2 := REAL_TO_INT_E(LDP(TRUE, If_Fruits_Ended), O_stock, _t1);
LT_E(_e2 AND LDP(TRUE, If_Fruits_Ended), _t1, Const2, _t3);
_e5 := MUL_E(LDP(TRUE, If_Fruits_Ended), C_Stock, O_stock, _t4);
_e7 := MUL_E(_e5 AND LDP(TRUE, If_Fruits_Ended), _t4, P_stock, _t6);
LE_E(_e7 AND LDP(TRUE, If_Fruits_Ended), _t6, Zero, _t8);
End_Day := _t3 OR LDP(TRUE, End_Day_007) OR End_Day OR _t8;
(* network 44 *)
(* איפוס מונים ונורות חיווי לקראת יום חדש *)
_p1 := LDP(TRUE, If_Fruits_Ended) OR LDP(TRUE, Start_Again);
_e2 := MOVE_E(_p1, Zero, P_C_Wash_Amount);
_e3 := MOVE_E(_e2, Zero, Half_Oranges);
_e4 := MOVE_E(_e3, Zero, Orange_AmountInWash);
MOVE_E(_e4, Zero, Juice_To_Filter);
_e5 := MOVE_E(_p1, Zero, allToSq);
_e6 := MOVE_E(_e5, Zero, Analog_Value);
_e7 := RST(_e6, Counting_Rates);
_e8 := RST(_e7, Total_Rates);
RST(_e8, Can_Start_Valid);
_e9 := RST(_p1, Click_Twice);
_e10 := RST(_e9, Counting_Input);
_e11 := RST(_e10, Val_Bool);
_e12 := RST(_e11, Validation_Check);
_e13 := RST(_e12, Analog_Showed);
RST(_e13, Stop_SqLight);
_e14 := RST(_p1, Input_In_Range);
_e15 := RST(_e14, Finished_5sec);
_e16 := RST(_e15, Start_5sec);
_e17 := RST(_e16, No_More);
RST(_e17, Storage_Filtered);
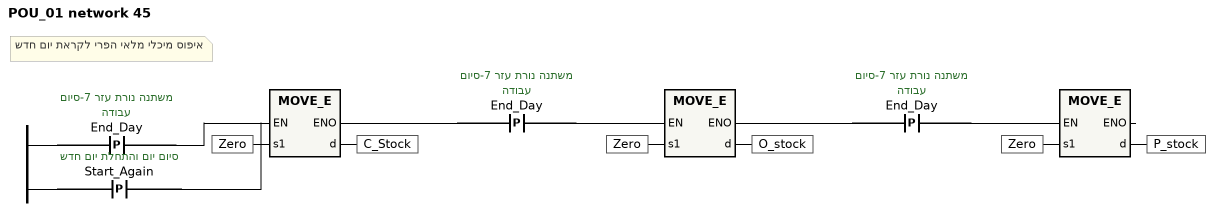
(* network 45 *)
(* איפוס מיכלי מלאי הפרי לקראת יום חדש *)
_e1 := MOVE_E(LDP(TRUE, End_Day) OR LDP(TRUE, Start_Again), Zero, C_Stock);
_e2 := MOVE_E(_e1 AND LDP(TRUE, End_Day), Zero, O_stock);
MOVE_E(_e2 AND LDP(TRUE, End_Day), Zero, P_stock);
END_PROGRAM
